FUNCTION_BLOCK FB_OutRobot_BoxMoveTurnTableToRoundBelt EXTENDS FB_ObjectBase_V2
VAR_INPUT
//    Execute    :BOOL;   // True : This prog will start.
//    Abort      :BOOL;   // True : This prog will be abort.
//    Reset      :BOOL;   // True : This prog will be reset.
//    ObjectName :STRING; // Set this fb name(About it's action)
	INPUT            			   : REFERENCE TO ST_InputTable;
	Cylinders					   : REFERENCE TO ARRAY[0..1] OF FB_Cylinder;
	Clips						   : REFERENCE TO ARRAY[0..1] OF FB_Cylinder;
	AutoMode_TurnTableToRoundBelt : st_AutoMode_ClampingBoxesJob;	
END_VAR

VAR_OUTPUT
//    Busy    :BOOL;        // True : This prog is running.
//    Done    :BOOL;        // True : Command has been executed.
//    Aborted :BOOL;        // True : This prog is aborted.
//    Error   :BOOL;        // True : This prog has an error.
//    ErrorID :UINT;       // Output ErrorID
//    Status  :T_MaxString; // Output this prog status by string(255bytes)
END_VAR

VAR
//    eState :E_MethodStatus_Basic;
//	uiExecutingStep : UDINT; // This var is used to been controll STATE_EXECUTING process.
//	uiResettingStep : UDINT;
//	uiAbortingStep : UDINT;
//	_Executed :BOOL; // Executing process completed.
//	_Error : BOOL; // FB has an error.
//	_ResetCompleted : BOOL; // FB resetting completed.
//	_AbortCompleted : BOOL; // FB aborting completed.
	//_Abort		: BOOL;
	strStatus	: STRING;
	uiResumeStep : UINT;
	tonTimeOut   :TON;
	tonTimeDelay   :TON;
	iWorkingIndex : INT;
	_UniqueErrorCode :STRING;	
	PickingPos	: ARRAY[0..1] OF ST_PositionTable;
	PlacingPos  : ARRAY[0..1] OF ST_PositionTable;
	bSyncPick	: BOOL;
	bSyncPlace	: BOOL;	
	UseA	: BOOL;
	UseB	: BOOL;
END_VAR

A00_BasicUnits();
SUPER^.A10_StateControl();

ACTION A00_BasicUnits:
tonTimeOut(PT:=T#15S);
tonTimeDelay(PT:=T#1.5s);
END_ACTION

METHOD GetModelState
VAR_OUTPUT
    xDone    :BOOL;
    xBusy    :BOOL;
    xError   :BOOL;
    xAborted :BOOL;
    iErrorID :UDINT;
	UniqueErrorCode : STRING;
END_VAR
xDone    := Done;
xBusy    := Busy;
xError   := Error;
xAborted := Abort;
iErrorID := ErrorID;
UniqueErrorCode := THIS^.UniqueErrorCode;
END_METHOD

METHOD GetName : STRING
GetName := ObjectName;
END_METHOD

METHOD PRIVATE M_CheckCommand : BOOL
VAR_INPUT
END_VAR

M_CheckCommand := true;
END_METHOD

METHOD PRIVATE M_GetWorkingConditions : BOOL
VAR_INPUT
END_VAR
//For rare box move , Boxes must place on same position , therefor only work with TargetPosition of ClipA

IF AutoMode_TurnTableToRoundBelt.ClampingInfo.UseClibA THEN
	PickingPos[0] :=FUN_GetPositionTableData('R',1,0);
	PlacingPos[0] :=FUN_GetPositionTableData('A',5,0);
	UseA := TRUE;
END_IF

IF AutoMode_TurnTableToRoundBelt.ClampingInfo.UseClibB THEN
	PickingPos[1] :=FUN_GetPositionTableData('R',2,1);
	PlacingPos[1] :=FUN_GetPositionTableData('A',6,1);
	UseB :=TRUE;
END_IF

IF PlacingPos[0].X_Pos =PlacingPos[1].X_Pos AND PlacingPos[0].Y_Pos = PlacingPos[1].Y_Pos AND UseA AND UseB THEN
		bSyncPlace:=TRUE;
	ELSE
		bSyncPlace:=FALSE;	
END_IF
IF PickingPos[0].X_Pos =PickingPos[1].X_Pos AND PickingPos[0].Y_Pos = PickingPos[1].Y_Pos AND UseA AND UseB THEN
		bSyncPick:=TRUE;
	ELSE
		bSyncPick:=FALSE;	
END_IF
END_METHOD

METHOD PRIVATE M_RecoveryAllObjects : BOOL
VAR_INPUT
END_VAR
VAR 
	i : INT;
END_VAR
FOR i:=0 TO 1 DO
	IF Clips[i].xError THEN
		Clips[i].M_Reset();
		ELSE
		Clips[i].M_Retract();		
	END_IF
	IF Cylinders[i].xError THEN
	Cylinders[i].M_Reset();	
	ELSE
	Cylinders[i].M_Retract();	
	END_IF
END_FOR

IF arAxisCtrl_gb[AxisNo.OutRobot_X].Admin.Axis.Status.Error THEN

	arAxisCtrl_gb[AxisNo.OutRobot_X].Admin.ClearError:= TRUE;
ELSE
	arAxisCtrl_gb[AxisNo.OutRobot_X].Admin.ClearError:= FALSE;
END_IF

IF arAxisCtrl_gb[AxisNo.OutRobot_Y].Admin.Axis.Status.Error THEN

	arAxisCtrl_gb[AxisNo.OutRobot_Y].Admin.ClearError:= TRUE;
ELSE
	arAxisCtrl_gb[AxisNo.OutRobot_Y].Admin.ClearError:= FALSE;
END_IF
END_METHOD

METHOD  M_STATE_ABORTED
VAR_INPUT
END_VAR
ERROR :=TRUE;
Busy    := FALSE;
Aborted := TRUE;
Status := strStatus;

IF NOT Execute THEN
	eSTATE:=STATE_RESETTING;
END_IF

IF Execute AND Reset THEN
//	uiExecutingStep :=uiResumeStep;
	eSTATE:=STATE_EXECUTING;
END_IF
END_METHOD

METHOD  M_STATE_ABORTING
VAR_INPUT
END_VAR
VAR
	
i : int;
	bCylinderCheck: BOOL;
END_VAR
CASE uiAbortingStep OF
	0 :
		bCylinderCheck:=TRUE;
		FOR i :=0 TO 1 DO		
	    	Cylinders[i].M_Reset();
			Cylinders[i].M_Retract();
			bCylinderCheck:=bCylinderCheck AND Cylinders[i].InRearPosition;	
		END_FOR
		IF bCylinderCheck THEN		
			uiAbortingStep:=9999;
		END_IF
	
	9999:	_AbortCompleted:=TRUE;
END_CASE

IF _AbortCompleted THEN	
	eSTATE :=STATE_ABORTED;
END_IF
END_METHOD

METHOD  M_STATE_DONE
VAR_INPUT
END_VAR
Busy 	:= FALSE;
Done	:=TRUE;

IF NOT Execute THEN
	eSTATE:=STATE_RESETTING;
END_IF
END_METHOD

METHOD  M_STATE_DORMANT
VAR_INPUT
END_VAR
Busy            := FALSE;
Done            := FALSE;
Aborted         := FALSE;
Error           := FALSE;
ErrorID         := 0;
Status          := '';
_ResetCompleted := FALSE;
_Error          := FALSE;
_Executed       := FALSE;
strStatus :='No Error';
uiExecutingStep :=uiResettingStep :=uiResumeStep :=0;
tonTimeOut.IN :=TRUE;
_UniqueErrorCode:='0';
iWorkingIndex :=0;
bSyncPick :=FALSE;
bSyncPlace := FALSE;
UseA := FALSE;
UseB :=FALSE;

IF Execute THEN
	eSTATE:=STATE_EXECUTING;
END_IF
END_METHOD

METHOD  M_STATE_ERROR
VAR_INPUT
END_VAR
ERROR   :=TRUE;
Busy	:=FALSE;
Status := strStatus;
IF NOT Execute THEN	
eSTATE:=STATE_RESETTING;
END_IF
END_METHOD

METHOD  M_STATE_EXECUTING
VAR_INPUT
END_VAR
VAR_INST
	

END_VAR

VAR
	bCylinderCheck : BOOL := TRUE;
END_VAR
Busy :=TRUE;

CASE uiExecutingStep OF
	

0: //Idle
	tonTimeDelay.IN :=FALSE;
	tonTimeOut.IN := FALSE;
	iWorkingIndex :=0;	
	M_GetWorkingConditions();
	M_RecoveryAllObjects();
	uiExecutingStep := 100;
	
100: //Check command
	IF M_CheckCommand()THEN	
		uiExecutingStep:=200;
	END_IF
	
200: // Check  boxes on turntable

	IF (UseA AND NOT INPUT.bTurnTable_R1Detect_Sensor) OR (UseB AND NOT INPUT.bTurnTable_R2Detect_Sensor) THEN
		_Error:=TRUE;
		strStatus :='Box Not on Turntable';
	ELSE
		IF UseA THEN
			iWorkingIndex :=0;
		ELSE
			iWorkingIndex :=1;	
		END_IF
		
		uiExecutingStep:=1000;	
	END_IF

	
1000: 
	// Move OutRobot to First clip picking	
	 	 
	arAxisCtrl_gb[AxisNo.OutRobot_X].PosMode.Position := PickingPos[iWorkingIndex].X_Pos;		
	arAxisCtrl_gb[AxisNo.OutRobot_Y].PosMode.Position := PickingPos[iWorkingIndex].Y_Pos;	
	uiExecutingStep:=1100;
		// todo : Check axes is moving
1100:
	// Check outRobot arrived
	IF		(arAxisStatus_gb[AxisNo.OutRobot_X].Admin._OpModeAck = ModePosAbs AND arAxisStatus_gb[AxisNo.OutRobot_X].Admin.CmdDone) 
	AND (arAxisStatus_gb[AxisNo.OutRobot_Y].Admin._OpModeAck = ModePosAbs AND arAxisStatus_gb[AxisNo.OutRobot_Y].Admin.CmdDone) 
	THEN
		tonTimeOut.IN := FALSE;
		uiExecutingStep:=1200;
	END_IF	
	tonTimeOut.IN := TRUE;
	IF tonTimeOut.Q THEN
		tonTimeOut.IN := FALSE;
		_Error :=TRUE;
		strStatus :='Robot move to picking position timeout';
	END_IF
	
1200: //Clip Down Pick	  
	bCylinderCheck := TRUE;
	Cylinders[iWorkingIndex].M_Extend();
	bCylinderCheck := Cylinders[iWorkingIndex].InFrontPosition AND bCylinderCheck;
	IF bSyncPick THEN
		Cylinders[1].M_Extend();
		bCylinderCheck := Cylinders[1].InFrontPosition AND bCylinderCheck;
	END_IF	
	 
	IF bCylinderCheck THEN
		tonTimeOut.IN := FALSE;
		uiExecutingStep:=1300;
	END_IF 
	tonTimeOut.IN := TRUE;
	IF tonTimeOut.Q THEN
		tonTimeOut.IN := FALSE;
		_Abort :=TRUE;
		strStatus :='Cylinder pick down timeout';
	END_IF
	
1300: // Clip close Pick
	bCylinderCheck := TRUE;
	Clips[iWorkingIndex].M_Extend();
	bCylinderCheck := Clips[iWorkingIndex].InFrontPosition AND bCylinderCheck;
	IF bSyncPick THEN
		Clips[1].M_Extend();
		bCylinderCheck := Clips[1].InFrontPosition AND bCylinderCheck;
	END_IF	
	 
	IF bCylinderCheck THEN
		tonTimeOut.IN := FALSE;
		uiExecutingStep:=1400;
	END_IF 
	
		tonTimeOut.IN := TRUE;
	IF tonTimeOut.Q THEN
		tonTimeOut.IN := FALSE;
		_Abort :=TRUE;
		strStatus :='clip pick close timeout';
	END_IF
	
1400: // Clip Up Pick
	bCylinderCheck := TRUE;
	Cylinders[iWorkingIndex].M_Retract();
	bCylinderCheck := Cylinders[iWorkingIndex].InRearPosition AND bCylinderCheck;
	IF bSyncPick THEN
		Cylinders[1].M_Retract();
		bCylinderCheck := Cylinders[1].InRearPosition AND bCylinderCheck;
	END_IF	
	 
	IF bCylinderCheck THEN
		tonTimeOut.IN := FALSE;
		uiExecutingStep:=1500;
	END_IF 
	
		tonTimeOut.IN := TRUE;
	IF tonTimeOut.Q THEN
		tonTimeOut.IN := FALSE;
		_Abort :=TRUE;
		strStatus :='cylinder pick up timeout';
	END_IF
	  
1500: // If Next pick
	  IF iWorkingIndex>=1 OR bSyncPick OR NOT UseB THEN
		//Go to placing step
			IF UseA THEN
				iWorkingIndex:=0;
			ELSE
				iWorkingIndex:=1;	
			END_IF
			uiExecutingStep:=1600;
		ELSE
			iWorkingIndex :=iWorkingIndex +1;
			uiExecutingStep:=1000;	
	  END_IF
	  
1600: // Check box
		
	IF (UseA AND  INPUT.bTurnTable_R1Detect_Sensor) OR (UseB AND  INPUT.bTurnTable_R2Detect_Sensor) THEN
		
		//
	ELSE
		tonTimeOut.IN := FALSE;
		uiExecutingStep:=2000;
	END_IF
		tonTimeOut.IN := TRUE;
	IF tonTimeOut.Q THEN
		tonTimeOut.IN := FALSE;
		_Error :=TRUE;
		strStatus :='Box still on Turntable';
	END_IF

2000: // Move to Placing pos	 
	 arAxisCtrl_gb[AxisNo.OutRobot_X].PosMode.Position := PlacingPos[iWorkingIndex].X_Pos;		
	 arAxisCtrl_gb[AxisNo.OutRobot_Y].PosMode.Position := PlacingPos[iWorkingIndex].Y_Pos;	
	 uiExecutingStep:=2100;

2100: // Waiting outRobot move to placing pos	 	
	 IF	(arAxisStatus_gb[AxisNo.OutRobot_X].Admin._OpModeAck = ModePosAbs AND arAxisStatus_gb[AxisNo.OutRobot_X].Admin.CmdDone) 
	AND (arAxisStatus_gb[AxisNo.OutRobot_Y].Admin._OpModeAck = ModePosAbs AND arAxisStatus_gb[AxisNo.OutRobot_Y].Admin.CmdDone)
	AND  tonTimeDelay.Q
	THEN		
		tonTimeOut.IN := FALSE;
		uiExecutingStep:=2200;
	END_IF	

		tonTimeOut.IN := TRUE;
	IF tonTimeOut.Q THEN
		tonTimeOut.IN := FALSE;
		_Error :=TRUE;
		strStatus :='robot move to placing position timeout';
	END_IF


2200: //Cllp Down place
	bCylinderCheck := TRUE;
	Cylinders[iWorkingIndex].M_Extend();
	bCylinderCheck := Cylinders[iWorkingIndex].InFrontPosition AND bCylinderCheck;
	IF bSyncPlace THEN
		Cylinders[1].M_Extend();
		bCylinderCheck := Cylinders[1].InFrontPosition AND bCylinderCheck;
	END_IF	
	 
	IF bCylinderCheck THEN
		tonTimeOut.IN := FALSE;
		uiExecutingStep:=2300;
	END_IF 
		tonTimeOut.IN := TRUE;
	IF tonTimeOut.Q THEN
		tonTimeOut.IN := FALSE;
		_Abort :=TRUE;
		strStatus :='Cylinder place down timeout';
	END_IF
	
2300: // Clip open Place
	bCylinderCheck := TRUE;
	Clips[iWorkingIndex].M_Retract();
	bCylinderCheck := Clips[iWorkingIndex].InRearPosition AND bCylinderCheck;
	IF bSyncPlace THEN
		Clips[1].M_Retract();
		bCylinderCheck := Clips[1].InRearPosition AND bCylinderCheck;
	END_IF	
	 
	IF bCylinderCheck THEN
		tonTimeOut.IN := FALSE;
		uiExecutingStep:=2400;
	END_IF 
	  
		tonTimeOut.IN := TRUE;
	IF tonTimeOut.Q THEN
		tonTimeOut.IN := FALSE;
		_Abort :=TRUE;
		strStatus :='clip place open timeout';
	END_IF
	  
2400: // Clip up Placing
	bCylinderCheck := TRUE;
	Cylinders[iWorkingIndex].M_Retract();
	bCylinderCheck := Cylinders[iWorkingIndex].InRearPosition AND bCylinderCheck;
	IF bSyncPlace THEN
		Cylinders[1].M_Retract();
		bCylinderCheck := Cylinders[1].InRearPosition AND bCylinderCheck;
	END_IF	
	 
	IF bCylinderCheck THEN
		tonTimeOut.IN := FALSE;
		uiExecutingStep:=2500;
	END_IF 
		tonTimeOut.IN := TRUE;
	IF tonTimeOut.Q THEN
		tonTimeOut.IN := FALSE;
		_Abort :=TRUE;
		strStatus :='cylinder place up timeout';
	END_IF
	
2500: // If Next place
	IF iWorkingIndex>=1 OR bSyncPlace OR NOT UseB THEN
		uiExecutingStep:=2600;
		// Finish
	ELSE	
		iWorkingIndex := iWorkingIndex+1;
	  	uiExecutingStep:=2000;
	END_IF
	
2600: // Finish	
	_Executed:=TRUE;
	
END_CASE
	
IF NOT Execute THEN
	eState:=STATE_RESETTING;
END_IF
IF _Error THEN
	eState:=STATE_ERROR;
END_IF
IF _Abort THEN
	eSTATE:=STATE_ABORTING;
END_IF
IF _Executed THEN
	eSTATE:=STATE_Done;
END_IF
END_METHOD

METHOD  M_STATE_RESETTING
VAR_INPUT
END_VAR
Error :=_Error;
Done :=_Executed;
Busy := FALSE;


CASE uiResettingStep OF
	
	0:
		M_RecoveryAllObjects();
		uiResettingStep:=9999;


	9999:
		_ResetCompleted:=TRUE;
END_CASE
IF _ResetCompleted THEN
	eSTATE:=STATE_DORMANT;
END_IF
END_METHOD

END_FUNCTION_BLOCK

(* stored: Version 1.1.0.1, ProductVersion 3.1.4024.13
   POU FB_OutRobot_BoxMoveTurnTableToRoundBelt: Id {c565a47a-9a73-42bd-ace5-577cda7be70e}, SpecialFunc None
   Folder Method: Id {54c021e8-903c-4c87-86d1-07bf3dcd049e}
   Folder STATE: Id {44c5b617-5355-4820-8843-0d57589ea95a}
   Action A00_BasicUnits: Id {f443de30-d582-456f-a66c-955d9cad232f}
   Method GetModelState: Id {b467df99-03ec-47c3-ad84-bf3ac65ce1ef}
   Method GetName: Id {a3ec3af2-b036-4a2c-a113-ff07b578e210}
   Method M_CheckCommand: Id {a29fac7b-4e8b-4642-8a60-a6f765b8d7a6}
   Method M_GetWorkingConditions: Id {6ae280d7-2ad1-464e-9b4c-3454ce766049}
   Method M_RecoveryAllObjects: Id {14e9b72e-6402-4009-9b41-438d9a88b60e}
   Method M_STATE_ABORTED: Id {d4845048-9779-4e6c-9fcf-93ce434ae95a}
   Method M_STATE_ABORTING: Id {93e90db1-874a-46ce-8d6b-c7c05e601fca}
   Method M_STATE_DONE: Id {6973f3fb-94b1-47a9-8b7c-13312ddece6d}
   Method M_STATE_DORMANT: Id {3d6f79a1-d758-494e-ab82-886c23f43abb}
   Method M_STATE_ERROR: Id {bc7653ad-6a09-4749-9e5e-a301806467ca}
   Method M_STATE_EXECUTING: Id {fa13af65-b2ec-40bb-8dbc-0297d8aad580}
   Method M_STATE_RESETTING: Id {5fc3bb5a-7008-45c2-b42f-391f35dcbf68} *)
